FUNCTION_BLOCK TFPalletizerGestione_PickPoint_Rulliere
(* Valorizza e aggiorna le variabili di stato del Pick-Point sulla base dei valori ricevuti dalla linea e dai valori inviati alla linea *)
VAR_INPUT
	WorkPickPoint : POINTER TO ARRAY [1..MAXPICKPOINT] OF TFMachinePalletizer_WorkPickPointSlab;
	WorkPickPointState : POINTER TO ARRAY [1..MAXPICKPOINT] OF TFMachinePalletizer_WorkPickPoint_State;
	WorkPickPointStateDaLinea : POINTER TO ARRAY [1..MAXPICKPOINT] OF TFMachinePalletizer_WorkPickPointRoller_State_DaLinea;
	WorkPickPointStateALinea : POINTER TO ARRAY [1..MAXPICKPOINT] OF TFMachinePalletizer_WorkPickPointRoller_State_ALinea;

END_VAR
VAR_OUTPUT
END_VAR
VAR
	wpp : INT;
END_VAR


FOR wpp:= 1 TO MAXPICKPOINT DO 
(******************* Valorizzazione da LINEA a PALLETTIZZATORE *********************)
	(* Set stato *)
	IF WorkPickPointStateDaLinea^[wpp].Automatico THEN
		WorkPickPointState^[wpp].State := WORKPICKPOINT_STATE_AUTO;
	ELSIF NOT WorkPickPointStateDaLinea^[wpp].Automatico THEN
		WorkPickPointState^[wpp].State := WORKPICKPOINT_STATE_MAN;
	ELSIF WorkPickPointStateDaLinea^[wpp].Errore THEN
		WorkPickPointState^[wpp].State := WORKPICKPOINT_STATE_ERROR;
	END_IF
	(* Set Marcia Presente/Assente *)
	IF WorkPickPointStateDaLinea^[wpp].PowerOK THEN
		WorkPickPointState^[wpp].PowerOK := TRUE;
	ELSE
		WorkPickPointState^[wpp].PowerOK := FALSE;
	END_IF
	(* Set Lastra Presente/Assente *)
	IF WorkPickPointStateDaLinea^[wpp].Occupato THEN
		WorkPickPointState^[wpp].ProdPresence := PROD_PRESENTE;
	ELSE
		WorkPickPointState^[wpp].ProdPresence := PROD_ASSENTE;
	END_IF
	(* Set Lastra Pronta/Non Pronta *)
	IF WorkPickPointStateDaLinea^[wpp].LastraPronta THEN
		WorkPickPointState^[wpp].LastraPronta := TRUE;
	ELSE
		WorkPickPointState^[wpp].LastraPronta := FALSE;
	END_IF
	(* Set CODICE *)
	WorkPickPointState^[wpp].Code := WorkPickPointStateDaLinea^[wpp].Codice; 
	(* Set Priorità *)
	IF WorkPickPointStateDaLinea^[wpp].Priority THEN
		WorkPickPointState^[wpp].Priority := MAX_PRIORITY;
	ELSE
		WorkPickPointState^[wpp].Priority := Min_PRIORITY;
	END_IF
	
(******************* Valorizzazione da PALLETTIZZATORE a LINEA *********************)	
	(* Set stato ingombro *)
	IF WorkPickPointState^[wpp].StatoIngombroEE = EE_IN_INGOMBRO THEN
		WorkPickPointStateALinea^[wpp].Ingombro 	:= TRUE;
	ELSIF WorkPickPointState^[wpp].StatoIngombroEE 	 = EE_FUORI_INGOMBRO THEN
		WorkPickPointStateALinea^[wpp].Ingombro 	:= FALSE;
	END_IF
	(* Set stato Prelievo *)
	IF WorkPickPointState^[wpp].StatoPrelievo = PRELIEVO_DA_EFFETTUARE THEN
		WorkPickPointStateALinea^[wpp].Prelievo_Effettuato := FALSE;
	ELSIF WorkPickPointState^[wpp].StatoPrelievo = PRELIEVO_EFFETTUATO THEN
		WorkPickPointStateALinea^[wpp].Prelievo_Effettuato := TRUE;
	END_IF

END_FOR

END_FUNCTION_BLOCK

(* stored: Version 1.1.0.1, ProductVersion 3.1.4024.11
   POU TFPalletizerGestione_PickPoint_Rulliere: Id {6b7f2e3a-6811-4036-8adc-b1d0325d64be}, SpecialFunc None *)
